INTERFACE ITF_pompdigin

METHOD get : bool
VAR_INPUT
	state : BOOL;
END_VAR
END_METHOD

END_INTERFACE

(* stored: Version 1.1.0.1, ProductVersion 3.1.4026.8
   Itf ITF_pompdigin: Id {885f5844-e201-4c58-87be-cb8e9c58d523}
   Method get: Id {610a700c-2748-4877-861d-6fd3abc371b2} *)
